TEXTLIST TL_E_CTRL_XPU
  0 = 'XTS_CMD_NULL'
  10 = 'XTS_CMD_INIT'
  30 = 'XTS_IDLE'
   = ''
END_TEXTLIST

(* stored: Version 1.1.0.1
   TextList TL_E_CTRL_XPU: Id {4a5412a8-9ab7-4150-87f1-6daf1a9346b4} *)
